// TIA Portal V20 export
TYPE "LER_typeEmRelation_Legacy"
// stored: Access Published, Namespace Unit1
   STRUCT
      emRelationEm_00 : "Unit1.LER_typeEmRelationEm_00";
      emRelationEm_01 : "Unit1.LER_typeEmRelationEm_01";
      emRelationEm_02 : "Unit1.LER_typeEmRelationEm_02";
      emRelationEm_03 : "Unit1.LER_typeEmRelationEm_03";
      emRelationEm_04 : "Unit1.LER_typeEmRelationEm_04";
      emRelationEm_05 : "Unit1.LER_typeEmRelationEm_05";
      emRelationEm_06 : "Unit1.LER_typeEmRelationEm_06";
      emRelationEm_07 : "Unit1.LER_typeEmRelationEm_07";
      emRelationEm_08 : "Unit1.LER_typeEmRelationEm_08";
      emRelationEm_09 : "Unit1.LER_typeEmRelationEm_09";
      emRelationEm_10 : "Unit1.LER_typeEmRelationEm_10";
      emRelationEm_11 : "Unit1.LER_typeEmRelationEm_11";
      emRelationEm_12 : "Unit1.LER_typeEmRelationEm_12";
      emRelationEm_13 : "Unit1.LER_typeEmRelationEm_13";
   END_STRUCT;
END_TYPE
